{attribute 'GeneratedUsingTerminal: EM7004-0000-0017'}
{attribute addProperty BoxType "EM7004-0000-0017"}
{attribute addProperty Id "StatusAT %I*Status_B4798D867Counter_valueAT %I*UINT2Latch_valueAT %I*UINT2"}
{attribute addProperty CRC "3853904169"}
{attribute addProperty Size "11"}
TYPE ENC_Inputs_Channel_E5B5E929 :
STRUCT
	{attribute addProperty Name "Status"}
	Status AT %I* : Status_B4798D86;
	{attribute addProperty Name "Counter_value"}
	Counter_value AT %I* : UINT;
	{attribute addProperty Name "Latch_value"}
	Latch_value AT %I* : UINT;
END_STRUCT
END_TYPE

(* stored: Version 1.2.0.0, ProductVersion 3.1.4024.9
   DUT ENC_Inputs_Channel_E5B5E929: Id {2ac74e88-9562-4e9d-a930-7823f9a08513} *)
